DATA_BLOCK "DB_SHO_Type"
TITLE =%version: 0.11 % CN: 20
//Function:
//
//Description:
//
//History:
//This version  %created_by:  nlhdl %
//              %date_created:  maandag 6 juli 2015 10:25:02 %
//              %release: VI_CONV/RA_Dev_Oakham %
//
//Modification History:                                   By:    Date:     Rev:
//----------------------------------------------------  -------  --------  -----
//7324: ECS-P General from the RD to RA for platform    nlHdL    06-07-15   0.11
//20085: ASI Slave errors on 62 and 63                  nltny    20-08-14   0.11
//18159: Add Fire Alarm Status                          nlMLaut  26-03-14   0.10
//15797: Keyword release added                          nlwwij   26-09-13   0.09
//14493: ASI Slave errors on 62 and 63                  nlHdL    02-07-13   0.08
//CR10485 Removed comment from type DB                  nlHHop   25-06-12   0.07
//CR7220 Changing SDS in SHO conform JES                nlple    04-07-11   0.06
//This is not a section, but an object                  nlJBax   01-04-11   0.05
//PR6177 Remove status change on HMI (No Error are WN)  nlHdL    05-01-11   0.04
//CR5712 Not used errors have number -1                 nlHdL    24-09-10   0.03
//CR5188 Updated to Coding conventions                  nlHdL    15-09-10   0.02
//Initial revision                                      insmahi  28-07-10   0.01
//
//
FAMILY : General
VERSION : 0.0


  STRUCT
   Type_Component : BYTE ;	//Type of the component (1 = Section, 0 = Other)
   Record_Length : BYTE ;	//Number of the Detailed Status in the UDT
   Status : ARRAY  [1 .. 32 ] OF "UDT_Comp_Status";
  END_STRUCT ;
BEGIN
   Type_Component := B#16#0;
   Record_Length := B#16#32;
   Status[1].HMI_Text_Number := -1;
   Status[1].Overall_Status_Relation := B#16#0;
   Status[1].General_Status_Relation := B#16#0;
   Status[2].HMI_Text_Number := -1;
   Status[2].Overall_Status_Relation := B#16#0;
   Status[2].General_Status_Relation := B#16#0;
   Status[3].HMI_Text_Number := -1;
   Status[3].Overall_Status_Relation := B#16#0;
   Status[3].General_Status_Relation := B#16#0;
   Status[4].HMI_Text_Number := -1;
   Status[4].Overall_Status_Relation := B#16#0;
   Status[4].General_Status_Relation := B#16#0;
   Status[5].HMI_Text_Number := -1;
   Status[5].Overall_Status_Relation := B#16#0;
   Status[5].General_Status_Relation := B#16#0;
   Status[6].HMI_Text_Number := -1;
   Status[6].Overall_Status_Relation := B#16#0;
   Status[6].General_Status_Relation := B#16#0;
   Status[7].HMI_Text_Number := -1;
   Status[7].Overall_Status_Relation := B#16#0;
   Status[7].General_Status_Relation := B#16#0;
   Status[8].HMI_Text_Number := -1;
   Status[8].Overall_Status_Relation := B#16#0;
   Status[8].General_Status_Relation := B#16#0;
   Status[9].HMI_Text_Number := 62;
   Status[9].Overall_Status_Relation := B#16#4;
   Status[9].General_Status_Relation := B#16#3;
   Status[10].HMI_Text_Number := 63;
   Status[10].Overall_Status_Relation := B#16#4;
   Status[10].General_Status_Relation := B#16#3;
   Status[11].HMI_Text_Number := 182;
   Status[11].Overall_Status_Relation := B#16#4;
   Status[11].General_Status_Relation := B#16#3;
   Status[12].HMI_Text_Number := 183;
   Status[12].Overall_Status_Relation := B#16#4;
   Status[12].General_Status_Relation := B#16#3;
   Status[13].HMI_Text_Number := 44;
   Status[13].Overall_Status_Relation := B#16#4;
   Status[13].General_Status_Relation := B#16#3;
   Status[14].HMI_Text_Number := 45;
   Status[14].Overall_Status_Relation := B#16#4;
   Status[14].General_Status_Relation := B#16#3;
   Status[15].HMI_Text_Number := 92;
   Status[15].Overall_Status_Relation := B#16#4;
   Status[15].General_Status_Relation := B#16#3;
   Status[16].HMI_Text_Number := 93;
   Status[16].Overall_Status_Relation := B#16#4;
   Status[16].General_Status_Relation := B#16#3;
   Status[17].HMI_Text_Number := -1;
   Status[17].Overall_Status_Relation := B#16#0;
   Status[17].General_Status_Relation := B#16#0;
   Status[18].HMI_Text_Number := -1;
   Status[18].Overall_Status_Relation := B#16#0;
   Status[18].General_Status_Relation := B#16#0;
   Status[19].HMI_Text_Number := 69;
   Status[19].Overall_Status_Relation := B#16#4;
   Status[19].General_Status_Relation := B#16#3;
   Status[20].HMI_Text_Number := 172;
   Status[20].Overall_Status_Relation := B#16#4;
   Status[20].General_Status_Relation := B#16#3;
   Status[21].HMI_Text_Number := 173;
   Status[21].Overall_Status_Relation := B#16#3;
   Status[21].General_Status_Relation := B#16#1;
   Status[22].HMI_Text_Number := 108;
   Status[22].Overall_Status_Relation := B#16#4;
   Status[22].General_Status_Relation := B#16#3;
   Status[23].HMI_Text_Number := 30;
   Status[23].Overall_Status_Relation := B#16#5;
   Status[23].General_Status_Relation := B#16#4;
   Status[24].HMI_Text_Number := -1;
   Status[24].Overall_Status_Relation := B#16#0;
   Status[24].General_Status_Relation := B#16#0;
   Status[25].HMI_Text_Number := -1;
   Status[25].Overall_Status_Relation := B#16#0;
   Status[25].General_Status_Relation := B#16#0;
   Status[26].HMI_Text_Number := -1;
   Status[26].Overall_Status_Relation := B#16#0;
   Status[26].General_Status_Relation := B#16#0;
   Status[27].HMI_Text_Number := -1;
   Status[27].Overall_Status_Relation := B#16#0;
   Status[27].General_Status_Relation := B#16#0;
   Status[28].HMI_Text_Number := -1;
   Status[28].Overall_Status_Relation := B#16#0;
   Status[28].General_Status_Relation := B#16#0;
   Status[29].HMI_Text_Number := -1;
   Status[29].Overall_Status_Relation := B#16#0;
   Status[29].General_Status_Relation := B#16#0;
   Status[30].HMI_Text_Number := -1;
   Status[30].Overall_Status_Relation := B#16#0;
   Status[30].General_Status_Relation := B#16#0;
   Status[31].HMI_Text_Number := -1;
   Status[31].Overall_Status_Relation := B#16#0;
   Status[31].General_Status_Relation := B#16#0;
   Status[32].HMI_Text_Number := -1;
   Status[32].Overall_Status_Relation := B#16#0;
   Status[32].General_Status_Relation := B#16#0;
END_DATA_BLOCK

